# EPICS substitutions: ek9000App/Db/EL3062.substitutions
file EL3062.template
{       pattern
        {
                TERMINAL,

        }
        {
        }
}
